TYPE ST_InputData_KL320x :
STRUCT
	usiState			: USINT;					//Input State from KL320x
	iDataIn				: INT;						//Input Data from KL320x
END_STRUCT
END_TYPE

(* stored: Version 1.1.0.1, ProductVersion 3.1.4024.6
   DUT ST_InputData_KL320x: Id {c824f9d9-f85d-4ef5-ab40-5b1159bb615d} *)
